// :Description: TcUnit suite for FB_Filter.
FUNCTION_BLOCK FB_FilterTests EXTENDS TcUnit.FB_TestSuite
VAR
    filter : FB_Filter;
    state  : E_State;
END_VAR


RollingAverage_passes_known_vector();


METHOD PRIVATE RollingAverage_passes_known_vector

TEST('RollingAverage_passes_known_vector');
AssertEquals_LREAL(Expected := 1.0, Actual := filter.Step(1.0), Delta := 0.001, Message := 'first sample');
TEST_FINISHED();
END_METHOD

END_FUNCTION_BLOCK

(* stored: Version 1.1.0.1, ProductVersion 3.1.4026.0
   POU FB_FilterTests: Id {bbbbbbbb-bbbb-bbbb-bbbb-bbbbbbbbbbb1}, SpecialFunc None
   Method RollingAverage_passes_known_vector: Id {bbbbbbbb-bbbb-bbbb-bbbb-bbbbbbbbbbb2} *)
